// TIA Portal V16 export
// export: Created 2021-12-01T21:20:02.5759828Z, ExportSetting WithDefaults, DisplayName Totally Integrated Automation Portal, DisplayVersion V16 Update 4, DisplayName TIA Portal Version Control Interface, DisplayVersion V16 Update 2, DisplayName TIA Portal Openness, DisplayVersion V16 Update 4, DisplayName SINAMICS Startdrive Advanced, DisplayVersion V16 Update 5, DisplayName SINAMICS Startdrive G130, G150, S120, S150, SINAMICS MV, S210, DisplayVersion V16 Update 5, DisplayName SINAMICS Startdrive G110M, G120, G120C, G120D, G120P, G115D, DisplayVersion V16 Update 5, DisplayName STEP 7 Professional, DisplayVersion V16 Update 4, DisplayName STEP 7 Safety, DisplayVersion V16, DisplayName WinCC Advanced, DisplayVersion V16 Update 4
FUNCTION "ST00262_1_FC" : Void   // FC123, LAD
TITLE = ST00262_1
{ S7_Optimized_Access := 'TRUE' }
VERSION : 0.1
// stored: AutoNumber true, IsIECCheckEnabled false, SetENOAutomatically false, UDAEnableTagReadback false
   VAR_IN_OUT
      OPMODE : "OPMODE_OUT_UDT";
      HMI_EXTENSION : "HMI_EXTENSION_PANEL_UDT";
   END_VAR
   VAR_TEMP
      EmptyHS : "RT_HANDSHAKE_UDT";
   END_VAR
BEGIN

REGION Network 1: Alarm
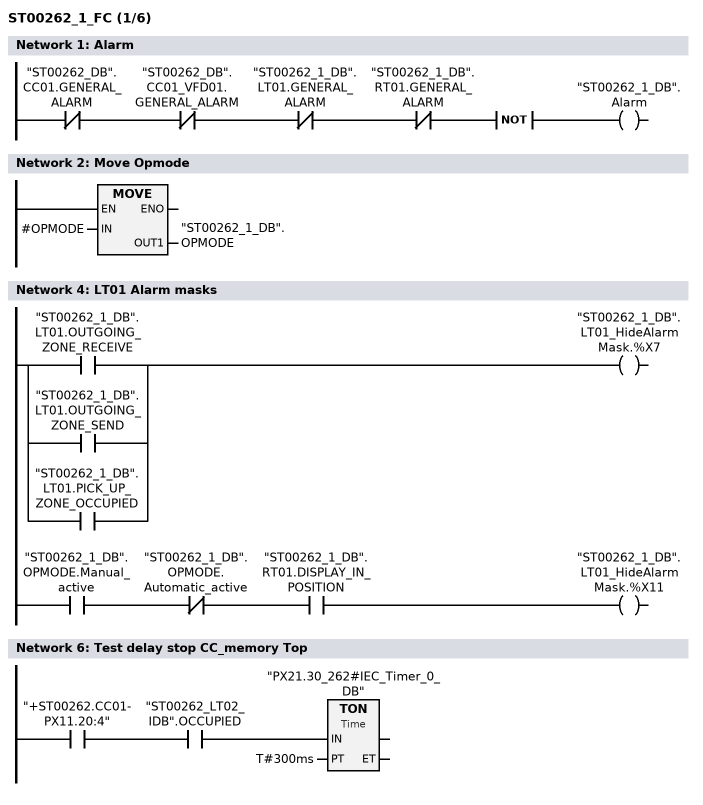
   RUNG wire#powerrail
      I_Contact( "ST00262_DB".CC01.GENERAL_ALARM )
      I_Contact( "ST00262_DB".CC01_VFD01.GENERAL_ALARM )
      I_Contact( "ST00262_1_DB".LT01.GENERAL_ALARM )
      I_Contact( "ST00262_1_DB".RT01.GENERAL_ALARM )
      Not()
      Coil( "ST00262_1_DB".Alarm )
   END_RUNG
   // the same network as SCL:
   "ST00262_1_DB".Alarm := NOT (NOT "ST00262_DB".CC01.GENERAL_ALARM AND NOT "ST00262_DB".CC01_VFD01.GENERAL_ALARM AND NOT "ST00262_1_DB".LT01.GENERAL_ALARM AND NOT "ST00262_1_DB".RT01.GENERAL_ALARM);
END_REGION

REGION Network 2: Move Opmode
   RUNG wire#powerrail
      Move(in := #OPMODE, out1 => "ST00262_1_DB".OPMODE)
   END_RUNG
   // the same network as SCL:
   "ST00262_1_DB".OPMODE := #OPMODE;
END_REGION

REGION Network 3: *******************LT01 Control*******************
END_REGION

REGION Network 4: LT01 Alarm masks
   RUNG wire#powerrail
      Contact( "ST00262_1_DB".LT01.OUTGOING_ZONE_RECEIVE )
      wire#w1
      Coil( "ST00262_1_DB".LT01_HideAlarmMask.%X7 )
   END_RUNG
   RUNG wire#powerrail
      Contact( "ST00262_1_DB".LT01.OUTGOING_ZONE_SEND )
   END_RUNG wire#w1
   RUNG wire#powerrail
      Contact( "ST00262_1_DB".LT01.PICK_UP_ZONE_OCCUPIED )
   END_RUNG wire#w1
   RUNG wire#powerrail
      Contact( "ST00262_1_DB".OPMODE.Manual_active )
      I_Contact( "ST00262_1_DB".OPMODE.Automatic_active )
      Contact( "ST00262_1_DB".RT01.DISPLAY_IN_POSITION )
      Coil( "ST00262_1_DB".LT01_HideAlarmMask.%X11 )
   END_RUNG
   // the same network as SCL:
   "ST00262_1_DB".LT01_HideAlarmMask.%X7 := "ST00262_1_DB".LT01.OUTGOING_ZONE_RECEIVE OR "ST00262_1_DB".LT01.OUTGOING_ZONE_SEND OR "ST00262_1_DB".LT01.PICK_UP_ZONE_OCCUPIED;
   "ST00262_1_DB".LT01_HideAlarmMask.%X11 := "ST00262_1_DB".OPMODE.Manual_active AND NOT "ST00262_1_DB".OPMODE.Automatic_active AND "ST00262_1_DB".RT01.DISPLAY_IN_POSITION;
END_REGION

REGION Network 5 (SCL): LT01 Parameters
   "ST00262_1_DB".LT01.PARA_SET.Para.HasMidPosition := false;
   "ST00262_1_DB".LT01.PARA_SET.Para.HasRT := true;
   "ST00262_1_DB".LT01.PARA_SET.Para.PosCCStopForward := true;
   "ST00262_1_DB".LT01.PARA_SET.Para.PosCCStopReverse := false;
   "ST00262_1_DB".LT01.PARA_SET.Para.PosRaiseForward_1 := true;
   "ST00262_1_DB".LT01.PARA_SET.Para.PosRaiseForward_2 := true;
   "ST00262_1_DB".LT01.PARA_SET.Para.PosRaiseReverse_1 := true;
   "ST00262_1_DB".LT01.PARA_SET.Para.PosRaiseReverse_2 := false;
   "ST00262_1_DB".LT01.PARA_SET.Para.PosSlowForward := true;
   "ST00262_1_DB".LT01.PARA_SET.Para.PosSlowReverse := false;
   "ST00262_1_DB".LT01.PARA_SET.Set.RuntimeLower := t#10s;
   "ST00262_1_DB".LT01.PARA_SET.Set.RuntimeLift := t#11s;
END_REGION

REGION Network 6: Test delay stop CC_memory Top
   RUNG wire#powerrail
      Contact( "+ST00262.CC01-PX11.20:4" )
      Contact( "ST00262_LT02_IDB".OCCUPIED )
      { S7_Templates := "time_type := Time" } "PX21.30_262#IEC_Timer_0_DB".TON(pt := T#300ms, et =>)
   END_RUNG
   // the same network as SCL:
   "PX21.30_262#IEC_Timer_0_DB".TON(IN := "+ST00262.CC01-PX11.20:4" AND "ST00262_LT02_IDB".OCCUPIED,
                           PT := T#300ms);
END_REGION

REGION Network 7: LT01 CC Place FB
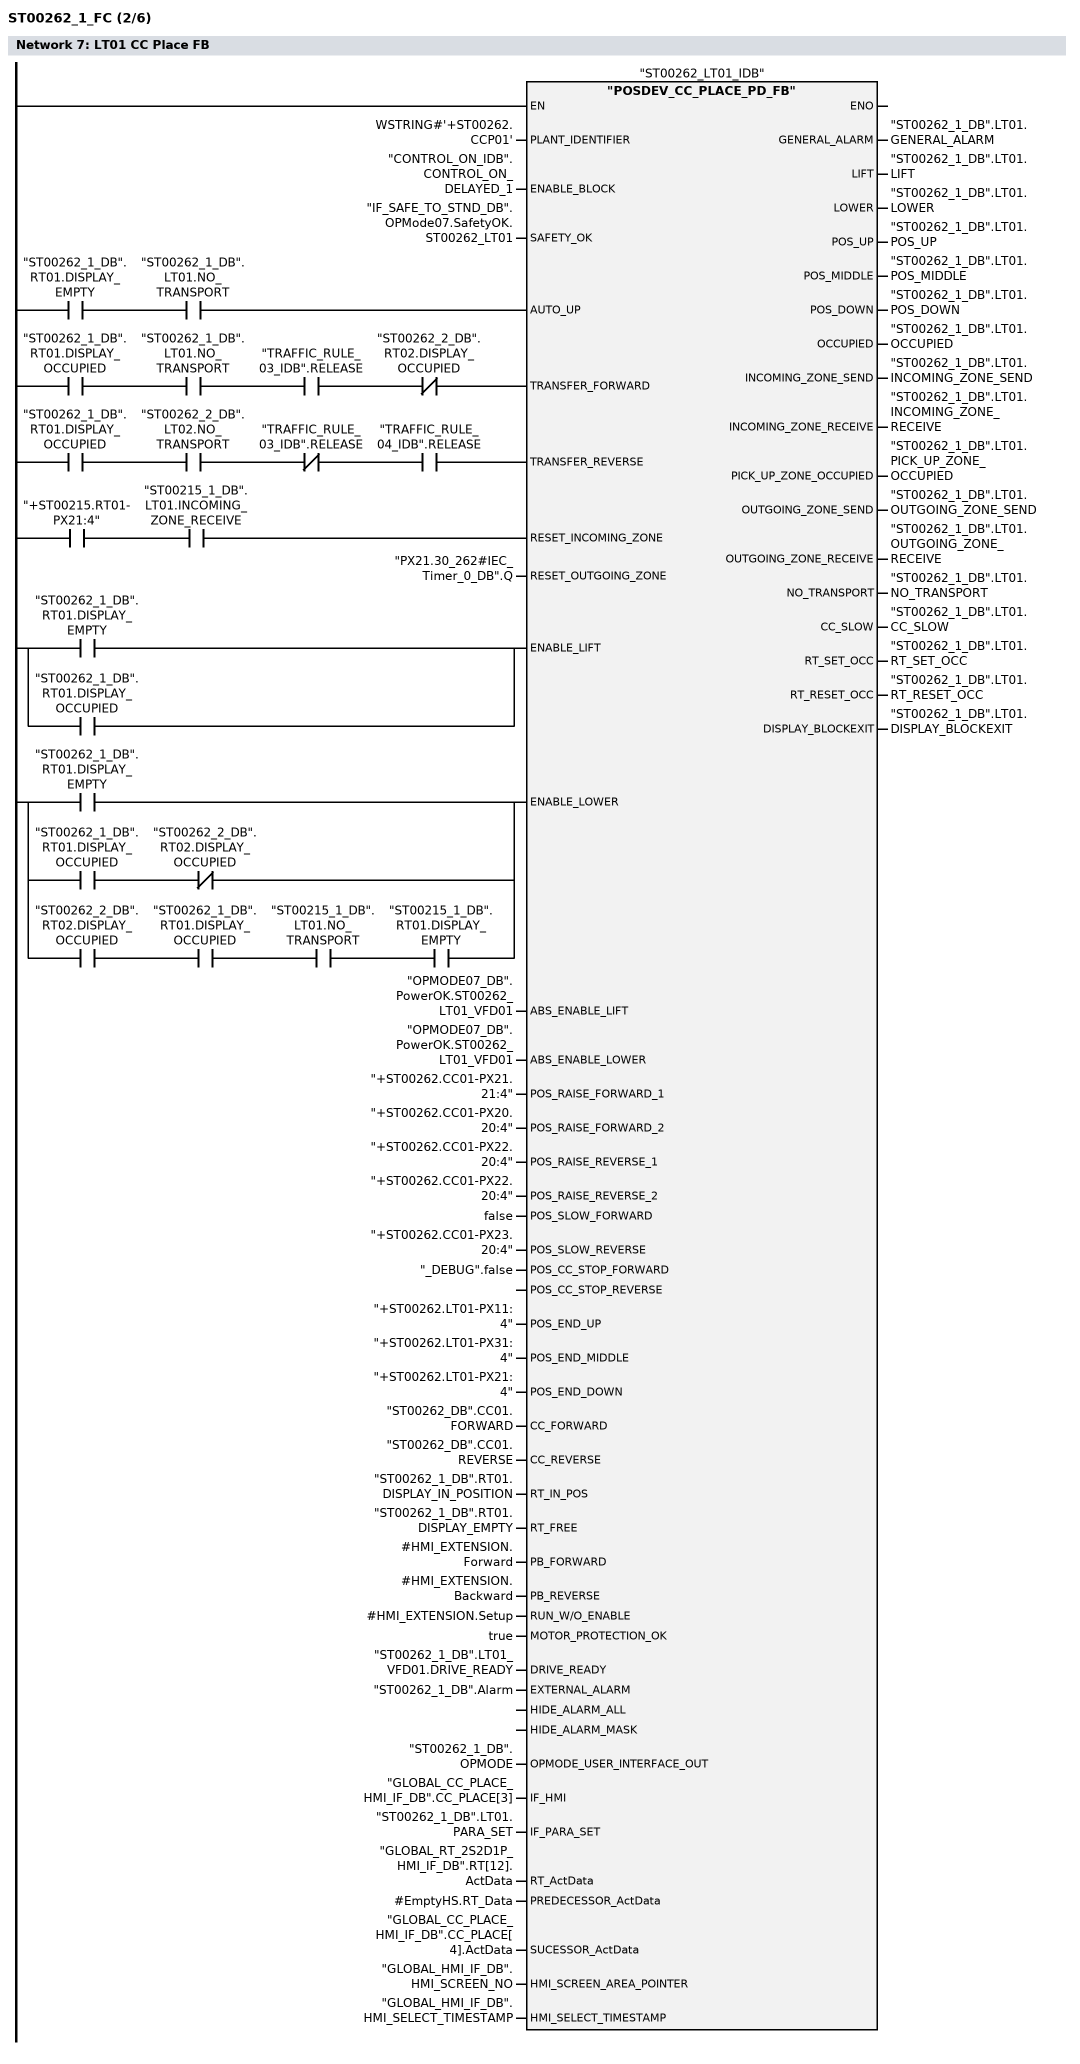
   RUNG wire#powerrail
      "ST00262_LT01_IDB"(AUTO_UP := wire#w1, TRANSFER_FORWARD := wire#w2, TRANSFER_REVERSE := wire#w3, RESET_INCOMING_ZONE := wire#w4, ENABLE_LIFT := wire#w5, ENABLE_LOWER := wire#w6, PLANT_IDENTIFIER := WSTRING#'+ST00262.CCP01', ENABLE_BLOCK := "CONTROL_ON_IDB".CONTROL_ON_DELAYED_1, SAFETY_OK := "IF_SAFE_TO_STND_DB".OPMode07.SafetyOK.ST00262_LT01, RESET_OUTGOING_ZONE := "PX21.30_262#IEC_Timer_0_DB".Q, ABS_ENABLE_LIFT := "OPMODE07_DB".PowerOK.ST00262_LT01_VFD01, ABS_ENABLE_LOWER := "OPMODE07_DB".PowerOK.ST00262_LT01_VFD01, POS_RAISE_FORWARD_1 := "+ST00262.CC01-PX21.21:4", POS_RAISE_FORWARD_2 := "+ST00262.CC01-PX20.20:4", POS_RAISE_REVERSE_1 := "+ST00262.CC01-PX22.20:4", POS_RAISE_REVERSE_2 := "+ST00262.CC01-PX22.20:4", POS_SLOW_FORWARD := false, POS_SLOW_REVERSE := "+ST00262.CC01-PX23.20:4", POS_CC_STOP_FORWARD := "_DEBUG".false, POS_CC_STOP_REVERSE :=, POS_END_UP := "+ST00262.LT01-PX11:4", POS_END_MIDDLE := "+ST00262.LT01-PX31:4", POS_END_DOWN := "+ST00262.LT01-PX21:4", CC_FORWARD := "ST00262_DB".CC01.FORWARD, CC_REVERSE := "ST00262_DB".CC01.REVERSE, RT_IN_POS := "ST00262_1_DB".RT01.DISPLAY_IN_POSITION, RT_FREE := "ST00262_1_DB".RT01.DISPLAY_EMPTY, PB_FORWARD := #HMI_EXTENSION.Forward, PB_REVERSE := #HMI_EXTENSION.Backward, "RUN_W/O_ENABLE" := #HMI_EXTENSION.Setup, MOTOR_PROTECTION_OK := true, DRIVE_READY := "ST00262_1_DB".LT01_VFD01.DRIVE_READY, EXTERNAL_ALARM := "ST00262_1_DB".Alarm, HIDE_ALARM_ALL :=, HIDE_ALARM_MASK :=, OPMODE_USER_INTERFACE_OUT := "ST00262_1_DB".OPMODE, IF_HMI := "GLOBAL_CC_PLACE_HMI_IF_DB".CC_PLACE[3], IF_PARA_SET := "ST00262_1_DB".LT01.PARA_SET, RT_ActData := "GLOBAL_RT_2S2D1P_HMI_IF_DB".RT[12].ActData, PREDECESSOR_ActData := #EmptyHS.RT_Data, SUCESSOR_ActData := "GLOBAL_CC_PLACE_HMI_IF_DB".CC_PLACE[4].ActData, HMI_SCREEN_AREA_POINTER := "GLOBAL_HMI_IF_DB".HMI_SCREEN_NO, HMI_SELECT_TIMESTAMP := "GLOBAL_HMI_IF_DB".HMI_SELECT_TIMESTAMP, GENERAL_ALARM => "ST00262_1_DB".LT01.GENERAL_ALARM, LIFT => "ST00262_1_DB".LT01.LIFT, LOWER => "ST00262_1_DB".LT01.LOWER, POS_UP => "ST00262_1_DB".LT01.POS_UP, POS_MIDDLE => "ST00262_1_DB".LT01.POS_MIDDLE, POS_DOWN => "ST00262_1_DB".LT01.POS_DOWN, OCCUPIED => "ST00262_1_DB".LT01.OCCUPIED, INCOMING_ZONE_SEND => "ST00262_1_DB".LT01.INCOMING_ZONE_SEND, INCOMING_ZONE_RECEIVE => "ST00262_1_DB".LT01.INCOMING_ZONE_RECEIVE, PICK_UP_ZONE_OCCUPIED => "ST00262_1_DB".LT01.PICK_UP_ZONE_OCCUPIED, OUTGOING_ZONE_SEND => "ST00262_1_DB".LT01.OUTGOING_ZONE_SEND, OUTGOING_ZONE_RECEIVE => "ST00262_1_DB".LT01.OUTGOING_ZONE_RECEIVE, NO_TRANSPORT => "ST00262_1_DB".LT01.NO_TRANSPORT, CC_SLOW => "ST00262_1_DB".LT01.CC_SLOW, RT_SET_OCC => "ST00262_1_DB".LT01.RT_SET_OCC, RT_RESET_OCC => "ST00262_1_DB".LT01.RT_RESET_OCC, DISPLAY_BLOCKEXIT => "ST00262_1_DB".LT01.DISPLAY_BLOCKEXIT)
   END_RUNG
   RUNG wire#powerrail
      Contact( "ST00262_1_DB".RT01.DISPLAY_EMPTY )
      Contact( "ST00262_1_DB".LT01.NO_TRANSPORT )
   END_RUNG wire#w1
   RUNG wire#powerrail
      Contact( "ST00262_1_DB".RT01.DISPLAY_OCCUPIED )
      Contact( "ST00262_1_DB".LT01.NO_TRANSPORT )
      Contact( "TRAFFIC_RULE_03_IDB".RELEASE )
      I_Contact( "ST00262_2_DB".RT02.DISPLAY_OCCUPIED )
   END_RUNG wire#w2
   RUNG wire#powerrail
      Contact( "ST00262_1_DB".RT01.DISPLAY_OCCUPIED )
      Contact( "ST00262_2_DB".LT02.NO_TRANSPORT )
      I_Contact( "TRAFFIC_RULE_03_IDB".RELEASE )
      Contact( "TRAFFIC_RULE_04_IDB".RELEASE )
   END_RUNG wire#w3
   RUNG wire#powerrail
      Contact( "+ST00215.RT01-PX21:4" )
      Contact( "ST00215_1_DB".LT01.INCOMING_ZONE_RECEIVE )
   END_RUNG wire#w4
   RUNG wire#powerrail
      Contact( "ST00262_1_DB".RT01.DISPLAY_EMPTY )
   END_RUNG wire#w5
   RUNG wire#powerrail
      Contact( "ST00262_1_DB".RT01.DISPLAY_OCCUPIED )
   END_RUNG wire#w5
   RUNG wire#powerrail
      Contact( "ST00262_1_DB".RT01.DISPLAY_EMPTY )
   END_RUNG wire#w6
   RUNG wire#powerrail
      Contact( "ST00262_1_DB".RT01.DISPLAY_OCCUPIED )
      I_Contact( "ST00262_2_DB".RT02.DISPLAY_OCCUPIED )
   END_RUNG wire#w6
   RUNG wire#powerrail
      Contact( "ST00262_2_DB".RT02.DISPLAY_OCCUPIED )
      Contact( "ST00262_1_DB".RT01.DISPLAY_OCCUPIED )
      Contact( "ST00215_1_DB".LT01.NO_TRANSPORT )
      Contact( "ST00215_1_DB".RT01.DISPLAY_EMPTY )
   END_RUNG wire#w6
   // the same network as SCL:
   "ST00262_LT01_IDB"(PLANT_IDENTIFIER := WSTRING#'+ST00262.CCP01',   // "POSDEV_CC_PLACE_PD_FB"
                      ENABLE_BLOCK := "CONTROL_ON_IDB".CONTROL_ON_DELAYED_1,
                      SAFETY_OK := "IF_SAFE_TO_STND_DB".OPMode07.SafetyOK.ST00262_LT01,
                      AUTO_UP := "ST00262_1_DB".RT01.DISPLAY_EMPTY AND "ST00262_1_DB".LT01.NO_TRANSPORT,
                      TRANSFER_FORWARD := "ST00262_1_DB".RT01.DISPLAY_OCCUPIED AND "ST00262_1_DB".LT01.NO_TRANSPORT AND "TRAFFIC_RULE_03_IDB".RELEASE AND NOT "ST00262_2_DB".RT02.DISPLAY_OCCUPIED,
                      TRANSFER_REVERSE := "ST00262_1_DB".RT01.DISPLAY_OCCUPIED AND "ST00262_2_DB".LT02.NO_TRANSPORT AND NOT "TRAFFIC_RULE_03_IDB".RELEASE AND "TRAFFIC_RULE_04_IDB".RELEASE,
                      RESET_INCOMING_ZONE := "+ST00215.RT01-PX21:4" AND "ST00215_1_DB".LT01.INCOMING_ZONE_RECEIVE,
                      RESET_OUTGOING_ZONE := "PX21.30_262#IEC_Timer_0_DB".Q,
                      ENABLE_LIFT := "ST00262_1_DB".RT01.DISPLAY_EMPTY OR "ST00262_1_DB".RT01.DISPLAY_OCCUPIED,
                      ENABLE_LOWER := "ST00262_1_DB".RT01.DISPLAY_EMPTY OR ("ST00262_1_DB".RT01.DISPLAY_OCCUPIED AND NOT "ST00262_2_DB".RT02.DISPLAY_OCCUPIED) OR ("ST00262_2_DB".RT02.DISPLAY_OCCUPIED AND "ST00262_1_DB".RT01.DISPLAY_OCCUPIED AND "ST00215_1_DB".LT01.NO_TRANSPORT AND "ST00215_1_DB".RT01.DISPLAY_EMPTY),
                      ABS_ENABLE_LIFT := "OPMODE07_DB".PowerOK.ST00262_LT01_VFD01,
                      ABS_ENABLE_LOWER := "OPMODE07_DB".PowerOK.ST00262_LT01_VFD01,
                      POS_RAISE_FORWARD_1 := "+ST00262.CC01-PX21.21:4",
                      POS_RAISE_FORWARD_2 := "+ST00262.CC01-PX20.20:4",
                      POS_RAISE_REVERSE_1 := "+ST00262.CC01-PX22.20:4",
                      POS_RAISE_REVERSE_2 := "+ST00262.CC01-PX22.20:4",
                      POS_SLOW_FORWARD := false,
                      POS_SLOW_REVERSE := "+ST00262.CC01-PX23.20:4",
                      POS_CC_STOP_FORWARD := "_DEBUG".false,
                      POS_END_UP := "+ST00262.LT01-PX11:4",
                      POS_END_MIDDLE := "+ST00262.LT01-PX31:4",
                      POS_END_DOWN := "+ST00262.LT01-PX21:4",
                      CC_FORWARD := "ST00262_DB".CC01.FORWARD,
                      CC_REVERSE := "ST00262_DB".CC01.REVERSE,
                      RT_IN_POS := "ST00262_1_DB".RT01.DISPLAY_IN_POSITION,
                      RT_FREE := "ST00262_1_DB".RT01.DISPLAY_EMPTY,
                      PB_FORWARD := #HMI_EXTENSION.Forward,
                      PB_REVERSE := #HMI_EXTENSION.Backward,
                      "RUN_W/O_ENABLE" := #HMI_EXTENSION.Setup,
                      MOTOR_PROTECTION_OK := true,
                      DRIVE_READY := "ST00262_1_DB".LT01_VFD01.DRIVE_READY,
                      EXTERNAL_ALARM := "ST00262_1_DB".Alarm,
                      OPMODE_USER_INTERFACE_OUT := "ST00262_1_DB".OPMODE,
                      IF_HMI := "GLOBAL_CC_PLACE_HMI_IF_DB".CC_PLACE[3],
                      IF_PARA_SET := "ST00262_1_DB".LT01.PARA_SET,
                      RT_ActData := "GLOBAL_RT_2S2D1P_HMI_IF_DB".RT[12].ActData,
                      PREDECESSOR_ActData := #EmptyHS.RT_Data,
                      SUCESSOR_ActData := "GLOBAL_CC_PLACE_HMI_IF_DB".CC_PLACE[4].ActData,
                      HMI_SCREEN_AREA_POINTER := "GLOBAL_HMI_IF_DB".HMI_SCREEN_NO,
                      HMI_SELECT_TIMESTAMP := "GLOBAL_HMI_IF_DB".HMI_SELECT_TIMESTAMP,
                      GENERAL_ALARM => "ST00262_1_DB".LT01.GENERAL_ALARM,
                      LIFT => "ST00262_1_DB".LT01.LIFT,
                      LOWER => "ST00262_1_DB".LT01.LOWER,
                      POS_UP => "ST00262_1_DB".LT01.POS_UP,
                      POS_MIDDLE => "ST00262_1_DB".LT01.POS_MIDDLE,
                      POS_DOWN => "ST00262_1_DB".LT01.POS_DOWN,
                      OCCUPIED => "ST00262_1_DB".LT01.OCCUPIED,
                      INCOMING_ZONE_SEND => "ST00262_1_DB".LT01.INCOMING_ZONE_SEND,
                      INCOMING_ZONE_RECEIVE => "ST00262_1_DB".LT01.INCOMING_ZONE_RECEIVE,
                      PICK_UP_ZONE_OCCUPIED => "ST00262_1_DB".LT01.PICK_UP_ZONE_OCCUPIED,
                      OUTGOING_ZONE_SEND => "ST00262_1_DB".LT01.OUTGOING_ZONE_SEND,
                      OUTGOING_ZONE_RECEIVE => "ST00262_1_DB".LT01.OUTGOING_ZONE_RECEIVE,
                      NO_TRANSPORT => "ST00262_1_DB".LT01.NO_TRANSPORT,
                      CC_SLOW => "ST00262_1_DB".LT01.CC_SLOW,
                      RT_SET_OCC => "ST00262_1_DB".LT01.RT_SET_OCC,
                      RT_RESET_OCC => "ST00262_1_DB".LT01.RT_RESET_OCC,
                      DISPLAY_BLOCKEXIT => "ST00262_1_DB".LT01.DISPLAY_BLOCKEXIT);
END_REGION

REGION Network 8: LT01 Speed
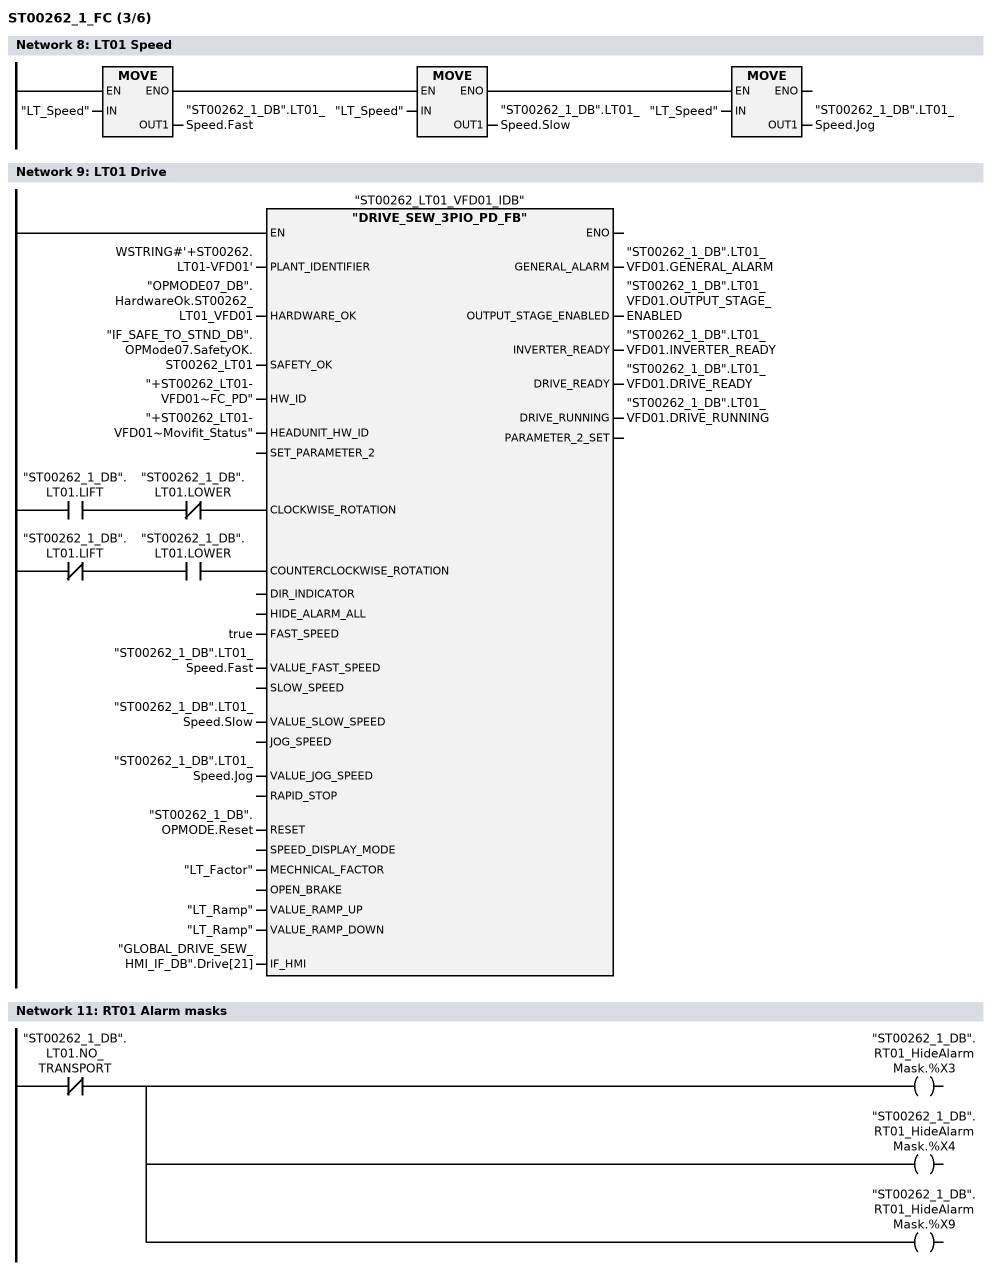
   RUNG wire#powerrail
      Move(in := "LT_Speed", out1 => "ST00262_1_DB".LT01_Speed.Fast)
      Move(in := "LT_Speed", out1 => "ST00262_1_DB".LT01_Speed.Slow)
      Move(in := "LT_Speed", out1 => "ST00262_1_DB".LT01_Speed.Jog)
   END_RUNG
   // the same network as SCL:
   "ST00262_1_DB".LT01_Speed.Fast := "LT_Speed";
   "ST00262_1_DB".LT01_Speed.Slow := "LT_Speed";
   "ST00262_1_DB".LT01_Speed.Jog := "LT_Speed";
END_REGION

REGION Network 9: LT01 Drive
   RUNG wire#powerrail
      "ST00262_LT01_VFD01_IDB"(CLOCKWISE_ROTATION := wire#w1, COUNTERCLOCKWISE_ROTATION := wire#w2, PLANT_IDENTIFIER := WSTRING#'+ST00262.LT01-VFD01', HARDWARE_OK := "OPMODE07_DB".HardwareOk.ST00262_LT01_VFD01, SAFETY_OK := "IF_SAFE_TO_STND_DB".OPMode07.SafetyOK.ST00262_LT01, HW_ID := "+ST00262_LT01-VFD01~FC_PD", HEADUNIT_HW_ID := "+ST00262_LT01-VFD01~Movifit_Status", SET_PARAMETER_2 :=, DIR_INDICATOR :=, HIDE_ALARM_ALL :=, FAST_SPEED := true, VALUE_FAST_SPEED := "ST00262_1_DB".LT01_Speed.Fast, SLOW_SPEED :=, VALUE_SLOW_SPEED := "ST00262_1_DB".LT01_Speed.Slow, JOG_SPEED :=, VALUE_JOG_SPEED := "ST00262_1_DB".LT01_Speed.Jog, RAPID_STOP :=, RESET := "ST00262_1_DB".OPMODE.Reset, SPEED_DISPLAY_MODE :=, MECHNICAL_FACTOR := "LT_Factor", OPEN_BRAKE :=, VALUE_RAMP_UP := "LT_Ramp", VALUE_RAMP_DOWN := "LT_Ramp", IF_HMI := "GLOBAL_DRIVE_SEW_HMI_IF_DB".Drive[21], GENERAL_ALARM => "ST00262_1_DB".LT01_VFD01.GENERAL_ALARM, OUTPUT_STAGE_ENABLED => "ST00262_1_DB".LT01_VFD01.OUTPUT_STAGE_ENABLED, INVERTER_READY => "ST00262_1_DB".LT01_VFD01.INVERTER_READY, DRIVE_READY => "ST00262_1_DB".LT01_VFD01.DRIVE_READY, DRIVE_RUNNING => "ST00262_1_DB".LT01_VFD01.DRIVE_RUNNING, PARAMETER_2_SET =>)
   END_RUNG
   RUNG wire#powerrail
      Contact( "ST00262_1_DB".LT01.LIFT )
      I_Contact( "ST00262_1_DB".LT01.LOWER )
   END_RUNG wire#w1
   RUNG wire#powerrail
      I_Contact( "ST00262_1_DB".LT01.LIFT )
      Contact( "ST00262_1_DB".LT01.LOWER )
   END_RUNG wire#w2
   // the same network as SCL:
   "ST00262_LT01_VFD01_IDB"(PLANT_IDENTIFIER := WSTRING#'+ST00262.LT01-VFD01',   // "DRIVE_SEW_3PIO_PD_FB"
                           HARDWARE_OK := "OPMODE07_DB".HardwareOk.ST00262_LT01_VFD01,
                           SAFETY_OK := "IF_SAFE_TO_STND_DB".OPMode07.SafetyOK.ST00262_LT01,
                           HW_ID := "+ST00262_LT01-VFD01~FC_PD",
                           HEADUNIT_HW_ID := "+ST00262_LT01-VFD01~Movifit_Status",
                           CLOCKWISE_ROTATION := "ST00262_1_DB".LT01.LIFT AND NOT "ST00262_1_DB".LT01.LOWER,
                           COUNTERCLOCKWISE_ROTATION := NOT "ST00262_1_DB".LT01.LIFT AND "ST00262_1_DB".LT01.LOWER,
                           FAST_SPEED := true,
                           VALUE_FAST_SPEED := "ST00262_1_DB".LT01_Speed.Fast,
                           VALUE_SLOW_SPEED := "ST00262_1_DB".LT01_Speed.Slow,
                           VALUE_JOG_SPEED := "ST00262_1_DB".LT01_Speed.Jog,
                           RESET := "ST00262_1_DB".OPMODE.Reset,
                           MECHNICAL_FACTOR := "LT_Factor",
                           VALUE_RAMP_UP := "LT_Ramp",
                           VALUE_RAMP_DOWN := "LT_Ramp",
                           IF_HMI := "GLOBAL_DRIVE_SEW_HMI_IF_DB".Drive[21],
                           GENERAL_ALARM => "ST00262_1_DB".LT01_VFD01.GENERAL_ALARM,
                           OUTPUT_STAGE_ENABLED => "ST00262_1_DB".LT01_VFD01.OUTPUT_STAGE_ENABLED,
                           INVERTER_READY => "ST00262_1_DB".LT01_VFD01.INVERTER_READY,
                           DRIVE_READY => "ST00262_1_DB".LT01_VFD01.DRIVE_READY,
                           DRIVE_RUNNING => "ST00262_1_DB".LT01_VFD01.DRIVE_RUNNING);
END_REGION

REGION Network 10: *******************RT01 Control*******************
END_REGION

REGION Network 11: RT01 Alarm masks
   RUNG wire#powerrail
      I_Contact( "ST00262_1_DB".LT01.NO_TRANSPORT )
      wire#w1
      Coil( "ST00262_1_DB".RT01_HideAlarmMask.%X3 )
   END_RUNG
   RUNG wire#w1
      Coil( "ST00262_1_DB".RT01_HideAlarmMask.%X4 )
   END_RUNG
   RUNG wire#w1
      Coil( "ST00262_1_DB".RT01_HideAlarmMask.%X9 )
   END_RUNG
   // the same network as SCL:
   "ST00262_1_DB".RT01_HideAlarmMask.%X3 := NOT "ST00262_1_DB".LT01.NO_TRANSPORT;
   "ST00262_1_DB".RT01_HideAlarmMask.%X4 := NOT "ST00262_1_DB".LT01.NO_TRANSPORT;
   "ST00262_1_DB".RT01_HideAlarmMask.%X9 := NOT "ST00262_1_DB".LT01.NO_TRANSPORT;
END_REGION

REGION Network 12 (SCL): RT01 Parameters
   "ST00262_1_DB".RT01.PARA_SET.Para.PosEndForward1 := true;
   "ST00262_1_DB".RT01.PARA_SET.Para.PosEndReverse := true;
   "ST00262_1_DB".RT01.PARA_SET.Para.PosSlowForward := true;

   "ST00262_1_DB".RT01.PARA_SET.Set.RunTimeForward := 450;
   "ST00262_1_DB".RT01.PARA_SET.Set.RunTimeReverse := 450;
END_REGION

REGION Network 13: RT01 HandShake
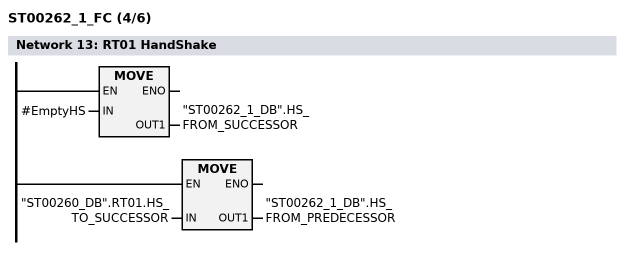
   RUNG wire#powerrail
      Move(in := #EmptyHS, out1 => "ST00262_1_DB".HS_FROM_SUCCESSOR)
   END_RUNG
   RUNG wire#powerrail
      Move(in := "ST00260_DB".RT01.HS_TO_SUCCESSOR, out1 => "ST00262_1_DB".HS_FROM_PREDECESSOR)
   END_RUNG
   // the same network as SCL:
   "ST00262_1_DB".HS_FROM_SUCCESSOR := #EmptyHS;
   "ST00262_1_DB".HS_FROM_PREDECESSOR := "ST00260_DB".RT01.HS_TO_SUCCESSOR;
END_REGION

REGION Network 14: RT01 FB Control
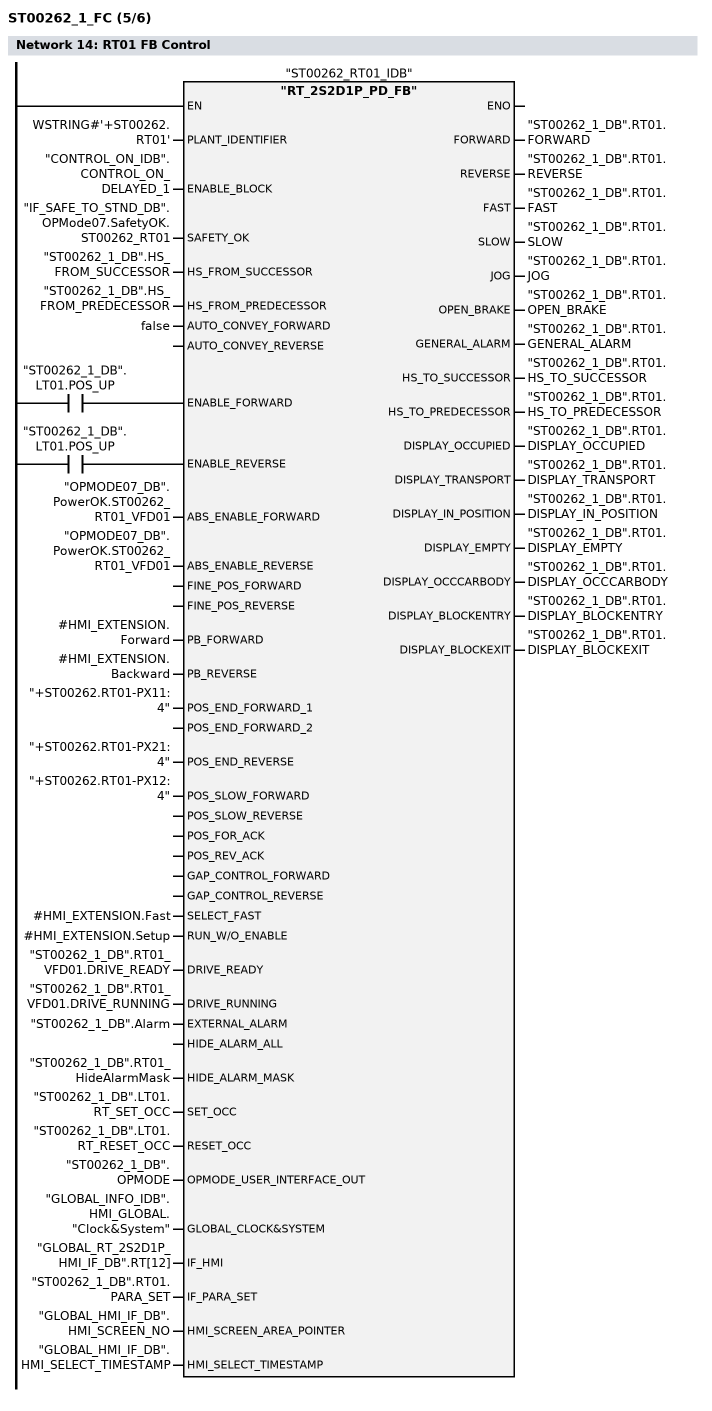
   RUNG wire#powerrail
      "ST00262_RT01_IDB"(ENABLE_FORWARD := wire#w1, ENABLE_REVERSE := wire#w2, PLANT_IDENTIFIER := WSTRING#'+ST00262.RT01', ENABLE_BLOCK := "CONTROL_ON_IDB".CONTROL_ON_DELAYED_1, SAFETY_OK := "IF_SAFE_TO_STND_DB".OPMode07.SafetyOK.ST00262_RT01, HS_FROM_SUCCESSOR := "ST00262_1_DB".HS_FROM_SUCCESSOR, HS_FROM_PREDECESSOR := "ST00262_1_DB".HS_FROM_PREDECESSOR, AUTO_CONVEY_FORWARD := false, AUTO_CONVEY_REVERSE :=, ABS_ENABLE_FORWARD := "OPMODE07_DB".PowerOK.ST00262_RT01_VFD01, ABS_ENABLE_REVERSE := "OPMODE07_DB".PowerOK.ST00262_RT01_VFD01, FINE_POS_FORWARD :=, FINE_POS_REVERSE :=, PB_FORWARD := #HMI_EXTENSION.Forward, PB_REVERSE := #HMI_EXTENSION.Backward, POS_END_FORWARD_1 := "+ST00262.RT01-PX11:4", POS_END_FORWARD_2 :=, POS_END_REVERSE := "+ST00262.RT01-PX21:4", POS_SLOW_FORWARD := "+ST00262.RT01-PX12:4", POS_SLOW_REVERSE :=, POS_FOR_ACK :=, POS_REV_ACK :=, GAP_CONTROL_FORWARD :=, GAP_CONTROL_REVERSE :=, SELECT_FAST := #HMI_EXTENSION.Fast, "RUN_W/O_ENABLE" := #HMI_EXTENSION.Setup, DRIVE_READY := "ST00262_1_DB".RT01_VFD01.DRIVE_READY, DRIVE_RUNNING := "ST00262_1_DB".RT01_VFD01.DRIVE_RUNNING, EXTERNAL_ALARM := "ST00262_1_DB".Alarm, HIDE_ALARM_ALL :=, HIDE_ALARM_MASK := "ST00262_1_DB".RT01_HideAlarmMask, SET_OCC := "ST00262_1_DB".LT01.RT_SET_OCC, RESET_OCC := "ST00262_1_DB".LT01.RT_RESET_OCC, OPMODE_USER_INTERFACE_OUT := "ST00262_1_DB".OPMODE, "GLOBAL_CLOCK&SYSTEM" := "GLOBAL_INFO_IDB".HMI_GLOBAL."Clock&System", IF_HMI := "GLOBAL_RT_2S2D1P_HMI_IF_DB".RT[12], IF_PARA_SET := "ST00262_1_DB".RT01.PARA_SET, HMI_SCREEN_AREA_POINTER := "GLOBAL_HMI_IF_DB".HMI_SCREEN_NO, HMI_SELECT_TIMESTAMP := "GLOBAL_HMI_IF_DB".HMI_SELECT_TIMESTAMP, FORWARD => "ST00262_1_DB".RT01.FORWARD, REVERSE => "ST00262_1_DB".RT01.REVERSE, FAST => "ST00262_1_DB".RT01.FAST, SLOW => "ST00262_1_DB".RT01.SLOW, JOG => "ST00262_1_DB".RT01.JOG, OPEN_BRAKE => "ST00262_1_DB".RT01.OPEN_BRAKE, GENERAL_ALARM => "ST00262_1_DB".RT01.GENERAL_ALARM, HS_TO_SUCCESSOR => "ST00262_1_DB".RT01.HS_TO_SUCCESSOR, HS_TO_PREDECESSOR => "ST00262_1_DB".RT01.HS_TO_PREDECESSOR, DISPLAY_OCCUPIED => "ST00262_1_DB".RT01.DISPLAY_OCCUPIED, DISPLAY_TRANSPORT => "ST00262_1_DB".RT01.DISPLAY_TRANSPORT, DISPLAY_IN_POSITION => "ST00262_1_DB".RT01.DISPLAY_IN_POSITION, DISPLAY_EMPTY => "ST00262_1_DB".RT01.DISPLAY_EMPTY, DISPLAY_OCCCARBODY => "ST00262_1_DB".RT01.DISPLAY_OCCCARBODY, DISPLAY_BLOCKENTRY => "ST00262_1_DB".RT01.DISPLAY_BLOCKENTRY, DISPLAY_BLOCKEXIT => "ST00262_1_DB".RT01.DISPLAY_BLOCKEXIT)
   END_RUNG
   RUNG wire#powerrail
      Contact( "ST00262_1_DB".LT01.POS_UP )
   END_RUNG wire#w1
   RUNG wire#powerrail
      Contact( "ST00262_1_DB".LT01.POS_UP )
   END_RUNG wire#w2
   // the same network as SCL:
   "ST00262_RT01_IDB"(PLANT_IDENTIFIER := WSTRING#'+ST00262.RT01',   // "RT_2S2D1P_PD_FB"
                      ENABLE_BLOCK := "CONTROL_ON_IDB".CONTROL_ON_DELAYED_1,
                      SAFETY_OK := "IF_SAFE_TO_STND_DB".OPMode07.SafetyOK.ST00262_RT01,
                      HS_FROM_SUCCESSOR := "ST00262_1_DB".HS_FROM_SUCCESSOR,
                      HS_FROM_PREDECESSOR := "ST00262_1_DB".HS_FROM_PREDECESSOR,
                      AUTO_CONVEY_FORWARD := false,
                      ENABLE_FORWARD := "ST00262_1_DB".LT01.POS_UP,
                      ENABLE_REVERSE := "ST00262_1_DB".LT01.POS_UP,
                      ABS_ENABLE_FORWARD := "OPMODE07_DB".PowerOK.ST00262_RT01_VFD01,
                      ABS_ENABLE_REVERSE := "OPMODE07_DB".PowerOK.ST00262_RT01_VFD01,
                      PB_FORWARD := #HMI_EXTENSION.Forward,
                      PB_REVERSE := #HMI_EXTENSION.Backward,
                      POS_END_FORWARD_1 := "+ST00262.RT01-PX11:4",
                      POS_END_REVERSE := "+ST00262.RT01-PX21:4",
                      POS_SLOW_FORWARD := "+ST00262.RT01-PX12:4",
                      SELECT_FAST := #HMI_EXTENSION.Fast,
                      "RUN_W/O_ENABLE" := #HMI_EXTENSION.Setup,
                      DRIVE_READY := "ST00262_1_DB".RT01_VFD01.DRIVE_READY,
                      DRIVE_RUNNING := "ST00262_1_DB".RT01_VFD01.DRIVE_RUNNING,
                      EXTERNAL_ALARM := "ST00262_1_DB".Alarm,
                      HIDE_ALARM_MASK := "ST00262_1_DB".RT01_HideAlarmMask,
                      SET_OCC := "ST00262_1_DB".LT01.RT_SET_OCC,
                      RESET_OCC := "ST00262_1_DB".LT01.RT_RESET_OCC,
                      OPMODE_USER_INTERFACE_OUT := "ST00262_1_DB".OPMODE,
                      "GLOBAL_CLOCK&SYSTEM" := "GLOBAL_INFO_IDB".HMI_GLOBAL."Clock&System",
                      IF_HMI := "GLOBAL_RT_2S2D1P_HMI_IF_DB".RT[12],
                      IF_PARA_SET := "ST00262_1_DB".RT01.PARA_SET,
                      HMI_SCREEN_AREA_POINTER := "GLOBAL_HMI_IF_DB".HMI_SCREEN_NO,
                      HMI_SELECT_TIMESTAMP := "GLOBAL_HMI_IF_DB".HMI_SELECT_TIMESTAMP,
                      FORWARD => "ST00262_1_DB".RT01.FORWARD,
                      REVERSE => "ST00262_1_DB".RT01.REVERSE,
                      FAST => "ST00262_1_DB".RT01.FAST,
                      SLOW => "ST00262_1_DB".RT01.SLOW,
                      JOG => "ST00262_1_DB".RT01.JOG,
                      OPEN_BRAKE => "ST00262_1_DB".RT01.OPEN_BRAKE,
                      GENERAL_ALARM => "ST00262_1_DB".RT01.GENERAL_ALARM,
                      HS_TO_SUCCESSOR => "ST00262_1_DB".RT01.HS_TO_SUCCESSOR,
                      HS_TO_PREDECESSOR => "ST00262_1_DB".RT01.HS_TO_PREDECESSOR,
                      DISPLAY_OCCUPIED => "ST00262_1_DB".RT01.DISPLAY_OCCUPIED,
                      DISPLAY_TRANSPORT => "ST00262_1_DB".RT01.DISPLAY_TRANSPORT,
                      DISPLAY_IN_POSITION => "ST00262_1_DB".RT01.DISPLAY_IN_POSITION,
                      DISPLAY_EMPTY => "ST00262_1_DB".RT01.DISPLAY_EMPTY,
                      DISPLAY_OCCCARBODY => "ST00262_1_DB".RT01.DISPLAY_OCCCARBODY,
                      DISPLAY_BLOCKENTRY => "ST00262_1_DB".RT01.DISPLAY_BLOCKENTRY,
                      DISPLAY_BLOCKEXIT => "ST00262_1_DB".RT01.DISPLAY_BLOCKEXIT);
END_REGION

REGION Network 15: RT01 Speed
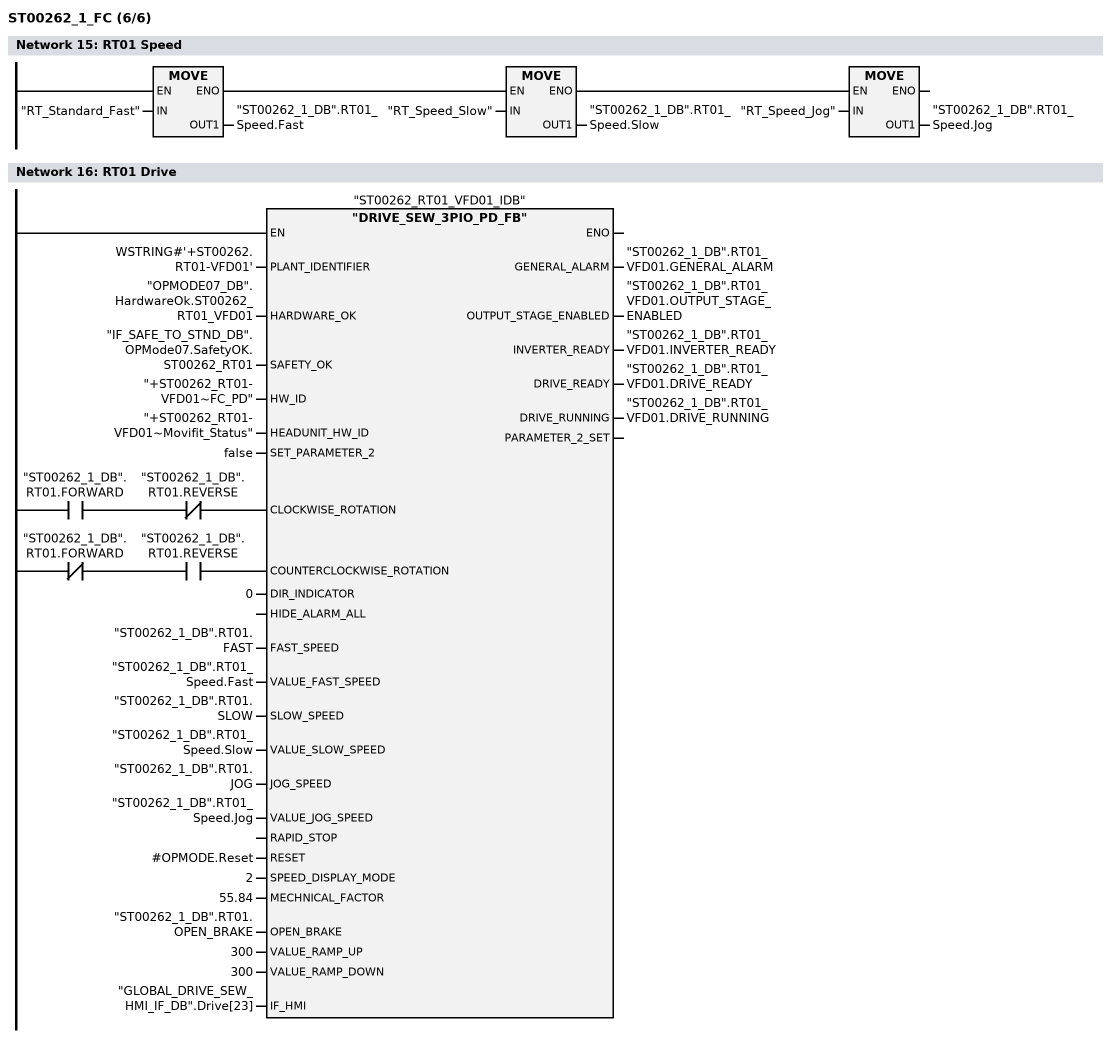
   RUNG wire#powerrail
      Move(in := "RT_Standard_Fast", out1 => "ST00262_1_DB".RT01_Speed.Fast)
      Move(in := "RT_Speed_Slow", out1 => "ST00262_1_DB".RT01_Speed.Slow)
      Move(in := "RT_Speed_Jog", out1 => "ST00262_1_DB".RT01_Speed.Jog)
   END_RUNG
   // the same network as SCL:
   "ST00262_1_DB".RT01_Speed.Fast := "RT_Standard_Fast";
   "ST00262_1_DB".RT01_Speed.Slow := "RT_Speed_Slow";
   "ST00262_1_DB".RT01_Speed.Jog := "RT_Speed_Jog";
END_REGION

REGION Network 16: RT01 Drive
   RUNG wire#powerrail
      "ST00262_RT01_VFD01_IDB"(CLOCKWISE_ROTATION := wire#w1, COUNTERCLOCKWISE_ROTATION := wire#w2, PLANT_IDENTIFIER := WSTRING#'+ST00262.RT01-VFD01', HARDWARE_OK := "OPMODE07_DB".HardwareOk.ST00262_RT01_VFD01, SAFETY_OK := "IF_SAFE_TO_STND_DB".OPMode07.SafetyOK.ST00262_RT01, HW_ID := "+ST00262_RT01-VFD01~FC_PD", HEADUNIT_HW_ID := "+ST00262_RT01-VFD01~Movifit_Status", SET_PARAMETER_2 := false, DIR_INDICATOR := 0, HIDE_ALARM_ALL :=, FAST_SPEED := "ST00262_1_DB".RT01.FAST, VALUE_FAST_SPEED := "ST00262_1_DB".RT01_Speed.Fast, SLOW_SPEED := "ST00262_1_DB".RT01.SLOW, VALUE_SLOW_SPEED := "ST00262_1_DB".RT01_Speed.Slow, JOG_SPEED := "ST00262_1_DB".RT01.JOG, VALUE_JOG_SPEED := "ST00262_1_DB".RT01_Speed.Jog, RAPID_STOP :=, RESET := #OPMODE.Reset, SPEED_DISPLAY_MODE := 2, MECHNICAL_FACTOR := 55.84, OPEN_BRAKE := "ST00262_1_DB".RT01.OPEN_BRAKE, VALUE_RAMP_UP := 300, VALUE_RAMP_DOWN := 300, IF_HMI := "GLOBAL_DRIVE_SEW_HMI_IF_DB".Drive[23], GENERAL_ALARM => "ST00262_1_DB".RT01_VFD01.GENERAL_ALARM, OUTPUT_STAGE_ENABLED => "ST00262_1_DB".RT01_VFD01.OUTPUT_STAGE_ENABLED, INVERTER_READY => "ST00262_1_DB".RT01_VFD01.INVERTER_READY, DRIVE_READY => "ST00262_1_DB".RT01_VFD01.DRIVE_READY, DRIVE_RUNNING => "ST00262_1_DB".RT01_VFD01.DRIVE_RUNNING, PARAMETER_2_SET =>)
   END_RUNG
   RUNG wire#powerrail
      Contact( "ST00262_1_DB".RT01.FORWARD )
      I_Contact( "ST00262_1_DB".RT01.REVERSE )
   END_RUNG wire#w1
   RUNG wire#powerrail
      I_Contact( "ST00262_1_DB".RT01.FORWARD )
      Contact( "ST00262_1_DB".RT01.REVERSE )
   END_RUNG wire#w2
   // the same network as SCL:
   "ST00262_RT01_VFD01_IDB"(PLANT_IDENTIFIER := WSTRING#'+ST00262.RT01-VFD01',   // "DRIVE_SEW_3PIO_PD_FB"
                           HARDWARE_OK := "OPMODE07_DB".HardwareOk.ST00262_RT01_VFD01,
                           SAFETY_OK := "IF_SAFE_TO_STND_DB".OPMode07.SafetyOK.ST00262_RT01,
                           HW_ID := "+ST00262_RT01-VFD01~FC_PD",
                           HEADUNIT_HW_ID := "+ST00262_RT01-VFD01~Movifit_Status",
                           SET_PARAMETER_2 := false,
                           CLOCKWISE_ROTATION := "ST00262_1_DB".RT01.FORWARD AND NOT "ST00262_1_DB".RT01.REVERSE,
                           COUNTERCLOCKWISE_ROTATION := NOT "ST00262_1_DB".RT01.FORWARD AND "ST00262_1_DB".RT01.REVERSE,
                           DIR_INDICATOR := 0,
                           FAST_SPEED := "ST00262_1_DB".RT01.FAST,
                           VALUE_FAST_SPEED := "ST00262_1_DB".RT01_Speed.Fast,
                           SLOW_SPEED := "ST00262_1_DB".RT01.SLOW,
                           VALUE_SLOW_SPEED := "ST00262_1_DB".RT01_Speed.Slow,
                           JOG_SPEED := "ST00262_1_DB".RT01.JOG,
                           VALUE_JOG_SPEED := "ST00262_1_DB".RT01_Speed.Jog,
                           RESET := #OPMODE.Reset,
                           SPEED_DISPLAY_MODE := 2,
                           MECHNICAL_FACTOR := 55.84,
                           OPEN_BRAKE := "ST00262_1_DB".RT01.OPEN_BRAKE,
                           VALUE_RAMP_UP := 300,
                           VALUE_RAMP_DOWN := 300,
                           IF_HMI := "GLOBAL_DRIVE_SEW_HMI_IF_DB".Drive[23],
                           GENERAL_ALARM => "ST00262_1_DB".RT01_VFD01.GENERAL_ALARM,
                           OUTPUT_STAGE_ENABLED => "ST00262_1_DB".RT01_VFD01.OUTPUT_STAGE_ENABLED,
                           INVERTER_READY => "ST00262_1_DB".RT01_VFD01.INVERTER_READY,
                           DRIVE_READY => "ST00262_1_DB".RT01_VFD01.DRIVE_READY,
                           DRIVE_RUNNING => "ST00262_1_DB".RT01_VFD01.DRIVE_RUNNING);
END_REGION
END_FUNCTION
